// TwinCAT 3 PLC project RT1
// ProgramVersion: 3.1.4026.16
// libraries:
//   Tc2_ControllerToolbox, * (Beckhoff Automation GmbH)
//   Tc2_Standard, * (Beckhoff Automation GmbH)
//   Tc2_System, * (Beckhoff Automation GmbH)
//   Tc2_Utilities, * (Beckhoff Automation GmbH)
//   Tc3_Module, * (Beckhoff Automation GmbH)
//   VisuDialogs, * (System)
// project tree:
//   / GlobalTextList.TcGTLO, PlcTask.TcTTO, Visualization Manager.TcVMO (not stored)
//   POUs/AuxFuns/ FB_AutoResetBool.TcPOU, FB_Blink.TcPOU, FB_INC_DEC_Integer.TcPOU, FB_RangeMonitor.TcPOU, prgTestAuxsFuns.TcPOU
//   POUs/Conversion/ F_DtToSqlTime.TcPOU, F_DtToSqlTime2.TcPOU, F_DtToStr.TcPOU, F_LrealToExcel.TcPOU, F_MatIdtoStr.TcPOU, F_TimeStToFileStr.TcPOU
//   POUs/CO_Ntrollers/ FB_BasicHist.TcPOU, PIController.TcPOU
//   POUs/Filters/ FB_AvgFilter.TcPOU (not stored), FB_SignalGen.TcPOU, prgFilterTesting.TcPOU
//   POUs/ MAIN.TcPOU
//   POUs/Math/ betwenLimits.TcPOU, CharCurve.TcPOU, CheckDivZero.TcPOU, Derivative.TcPOU, DerivativeFiltered.TcPOU, DerivativeFiltered_2.TcPOU, FB_CalcKeyPoints.TcPOU, FB_CalcPeriod.TcPOU, FB_RampReal.TcPOU, FB_RMSCalc.TcPOU, FB_TimeBasedIntegrator.TcPOU, FB_TimeCounter.TcPOU, FirstDegResponse.TcPOU, F_AdjustDecimals.TcPOU, F_AdjustPrecision.TcPOU, F_SimpleDeadBand.TcPOU, GVL_Math.TcGVL, Integral.TcPOU, LinTrafoLimitLess.TcPOU, LinTrafo_1.TcPOU, prgMathTesting.TcPOU, SawTooth.TcPOU, TriangleWave.TcPOU
//   POUs/OrderAlgorithms/ F_SortBubble.TcPOU, F_SortInsertion.TcPOU
//   POUs/SignalCalc/ FB_RmsCalc2.TcPOU
//   POUs/SpecialTriggers/ FB_ChangeTrig.TcPOU, FB_Int_Trig.TcPOU, FB_Int_TrigFall.TcPOU, FB_Int_TrigRise.TcPOU, prgTrigTesting.TcPOU
//   POUs/Statistics/ FB_BasicStatsFuns.TcPOU, prgTestStatistics.TcPOU
//   VISUs/AuxScreens/ Footer.TcVIS
//   VISUs/ Math.TcVIS, Visualization.TcVIS
// real-time tasks:
//   TASK PlcTask: cycle T#10ms, priority 20, ADS port 350

CONFIGURATION RT1
    RESOURCE PLC ON TwinCAT3
        TASK PlcTask(INTERVAL := T#10ms, PRIORITY := 20);
        PROGRAM MAIN WITH PlcTask : MAIN;
    END_RESOURCE
END_CONFIGURATION

// ---- POUs/Math/GVL_Math.TcGVL
{attribute 'qualified_only'}
VAR_GLOBAL PERSISTENT
	rIntegratorResult:LREAL;
END_VAR

// ---- POUs/MAIN.TcPOU
PROGRAM MAIN
VAR

	sinGen:FB_CTRL_SIGNAL_GENERATOR;
	mode: Tc2_ControllerToolbox.E_CTRL_MODE := Tc2_ControllerToolbox.E_CTRL_MODE.eCTRL_MODE_ACTIVE;
	sine: LREAL;
	paramSin: Tc2_ControllerToolbox.ST_CTRL_SIGNAL_GENERATOR_PARAMS := (tCtrlCycleTime := TIME#10MS, tTaskCycleTime := TIME#10MS, eSignalType := E_CTRL_SIGNAL_TYPE.eCTRL_SINUS, tCylceDuration := TIME#500MS, fAmplitude := 2);
	rms1: FB_RMSCalc;
	rms2: FB_RmsCalc2;
	rmsOut1: LREAL;
	rmsOut2: LREAL;
	bResetRms: BOOL;
	rPeriod: LREAL := 1;
END_VAR

prgTrigTesting();
prgTestAuxsFuns();
prgTestStatistics();
prgFilterTesting();
prgMathTesting();


sinGen(
	fManValue:= , 
	eMode:=mode , 
	fOut=> sine, 
	eState=> , 
	eErrorId=> , 
	bError=> , 
	stParams:= paramSin);
	


rms1(
	rInput:= sine, 
	rPastTime:= 0.01, 
	bReset:= bResetRms, 
	rPeriod:=rPeriod , 
	rRmsValue=> rmsOut1);
	
rms2(in:= sine, timePerCycle:= 0.01, result=> rmsOut2);

END_PROGRAM

// ---- POUs/Math/FB_RMSCalc.TcPOU
FUNCTION_BLOCK FB_RMSCalc
VAR_INPUT
	rInput:LREAL;
	rPastTime:LREAL;
	bReset: BOOL;
	rPeriod: LREAL;
END_VAR
VAR_OUTPUT
	rRmsValue:LREAL;
END_VAR
VAR
	rmsIntegral:Integral;
END_VAR
(*Bloco funcional calcula o valor RMS de uma onda senoidal*)
(*Ha limitacoes quanto à frequencia utilizada (os testes foram feitos com frequencias de ate 12hz)*)
(*e quanto ao scan do plc (task de 2ms, mais baixas apresentam problemas)*)

IF bReset THEN
	rRmsValue:=SQRT(1/rPeriod *(rmsIntegral.rIntegral));
END_IF
rmsIntegral(rInput:=EXPT(rInput,2),rPastTime:=rPastTime , bReset:=bReset);

END_FUNCTION_BLOCK

// ---- POUs/Math/Integral.TcPOU
FUNCTION_BLOCK Integral
VAR_INPUT
	rInput:LREAL;		(*Valor de entrada*)
	rPastTime:LREAL;	(*tempo decorrido em Seg*)
	bReset: BOOL;	(*reinicia o bloco da integral*)
END_VAR
VAR_OUTPUT
	rIntegral:LREAL;	(*integral calculada*)
END_VAR
VAR
	rOldIntegral: LREAL;	(*Ultimo valor da integral*)
END_VAR
(*Este bloco funcional calcula a integral de uma funcao*)

IF bReset THEN
	rIntegral:=0;
	rOldIntegral:=0;
ELSE
	rIntegral:=rPastTime*rInput+rOldIntegral;
END_IF
rOldIntegral:=rIntegral;

END_FUNCTION_BLOCK

// ---- POUs/SignalCalc/FB_RmsCalc2.TcPOU
FUNCTION_BLOCK FB_RmsCalc2
VAR_INPUT
	in:LREAL;				//input sinal to calculate rms value
	timePerCycle:LREAL;		//time per cycle in seconds
END_VAR
VAR_OUTPUT
	result:LREAL;
END_VAR
VAR
	ar:ARRAY[1..100] OF LREAL;
	i: INT;
	sum,mean,t:LREAL;
END_VAR

FOR i:= 100 TO 2 BY -1 DO
	ar[i]:= ar[i-1];
END_FOR
ar[1]:=in;
sum:=0;

FOR i:= 1 TO 100 DO
	sum:=sum + EXPT(ar[i],2);
END_FOR
mean:= sum/100;
t:=100*timePerCycle;
result:= SQRT((1/t)*mean);

END_FUNCTION_BLOCK

// ---- POUs/SpecialTriggers/prgTrigTesting.TcPOU
PROGRAM prgTrigTesting
VAR
	changeTrig1:FB_ChangeTrig;
	udi:UDINT:=10;
	udiTrigCnt:UDINT;
	changeTrig2:FB_ChangeTrig;
	r1:REAL:=10;
	r1TrigCnt2:UDINT;
	changeTrigStr:FB_ChangeTrig;
	s1:STRING:='Boa tarde';
	sTringCnt:UDINT;
END_VAR

IF changeTrig1.M_ChngTrig(udi) THEN
	udiTrigCnt:=udiTrigCnt+1;
END_IF
IF changeTrig2.M_ChngTrig(in:= r1) THEN
	r1TrigCnt2:=r1TrigCnt2+1;
END_IF
IF changeTrigStr.M_ChngTrig(s1) THEN
	sTringcnt:=sTringcnt+1;
END_IF

END_PROGRAM

// ---- POUs/SpecialTriggers/FB_ChangeTrig.TcPOU
FUNCTION_BLOCK FB_ChangeTrig
VAR_INPUT
END_VAR
VAR_OUTPUT
END_VAR
VAR
	internalPointer:POINTER TO BYTE;
	aBytes:ARRAY[0..254] OF BYTE;
END_VAR

METHOD M_ChngTrig : BOOL
VAR_INPUT
	in:ANY;
END_VAR
IF THIS^.internalPointer <> 0 THEN
	M_ChngTrig:= memcmp(in.pValue,THIS^.internalPointer, in.diSize) <> 0;
	memcpy(THIS^.internalPointer,in.pValue,in.diSize);
ELSE
	THIS^.internalPointer:= ADR(THIS^.aBytes);
END_IF
END_METHOD

END_FUNCTION_BLOCK

// ---- POUs/AuxFuns/prgTestAuxsFuns.TcPOU
PROGRAM prgTestAuxsFuns
VAR
	blink:FB_Blink;
	rBlinkOn:LREAL:=0.5;
	rBlinkOff:LREAL:=0.3;
	bOutputBlink: BOOL;
END_VAR

blink(tON:= LREAL_TO_TIME(rBlinkOn*1000), tOff:=LREAL_TO_TIME(rBlinkOff*1000) , output=> bOutputBlink);

END_PROGRAM

// ---- POUs/AuxFuns/FB_Blink.TcPOU
FUNCTION_BLOCK FB_Blink
VAR_INPUT
	tON,tOff:TIME;
END_VAR
VAR_OUTPUT
	output:BOOL;
END_VAR
VAR
	timer:ton;
END_VAR

timer(IN:=NOT timer.Q);
IF timer.Q THEN
	IF output THEN
		timer.PT:=tOff;
	ELSE
		timer.PT:=tOn;
	END_IF
	output:= NOT output;
END_IF

END_FUNCTION_BLOCK

// ---- POUs/Statistics/prgTestStatistics.TcPOU
PROGRAM prgTestStatistics
VAR
	statistics:FB_BasicStatsFuns;
	aStats: ARRAY [1..7] OF LREAL := [15, 12, 11, 7, -5, 33, 45];
	avg: LREAL;
	maxi: LREAL;
	mini: LREAL;
	range: LREAL;
	variance: LREAL;
	std:LREAL;
END_VAR

avg:= statistics.M_Avg(aStats);

maxi:=statistics.M_Max(aStats);

mini:= statistics.M_Min(aStats);

range:= statistics.M_Range(aStats);

variance:=statistics.M_Variance(aStats);

std:= statistics.M_Std(aStats);

END_PROGRAM

// ---- POUs/Statistics/FB_BasicStatsFuns.TcPOU
FUNCTION_BLOCK FB_BasicStatsFuns
VAR_INPUT
END_VAR
VAR_OUTPUT
END_VAR
VAR
END_VAR

METHOD M_Avg : LREAL
VAR_IN_OUT
	a : ARRAY[*] OF LREAL;
END_VAR

VAR
	upper: DINT;
	lower: DINT;
	sum:LREAL;
	idx:DINT;
	qtt: LREAL;
	avg: LREAL;
END_VAR
upper:=UPPER_BOUND(a,1);
lower:=LOWER_BOUND(a,1);

qtt:= DINT_TO_LREAL(upper-lower+1);

sum:=0;
FOR idx:=lower TO upper DO
	sum:= sum + a[idx];
END_FOR
IF qtt <> 0 THEN
	avg:= sum/qtt;
END_IF
M_Avg:=avg;
END_METHOD

METHOD M_Max : LREAL
VAR_IN_OUT
	a:ARRAY[*] OF LREAL;
END_VAR
VAR
	maximum:LREAL;
	upper: DINT;
	lower: DINT;
	range: LREAL;
	idx: DINT;
END_VAR
upper:=UPPER_BOUND(a,1);
lower:=LOWER_BOUND(a,1);

range:= DINT_TO_LREAL(upper-lower+1);

maximum:= a[lower];

FOR idx:= lower TO upper DO
	maximum:= MAX(maximum, a[idx]);
END_FOR
M_Max:= maximum;
END_METHOD

METHOD M_Min : LREAL
VAR_IN_OUT
	a:ARRAY[*] OF LREAL;
END_VAR
VAR
	minimum:LREAL;
	upper: DINT;
	lower: DINT;
	range: LREAL;
	idx: DINT;	
END_VAR
upper:=UPPER_BOUND(a,1);
lower:=LOWER_BOUND(a,1);

range:= DINT_TO_LREAL(upper-lower+1);

minimum:= a[lower];

FOR idx:= lower TO upper DO
	minimum:= MIN(minimum, a[idx]);
END_FOR
M_Min:= minimum;
END_METHOD

METHOD M_Range : LREAL
VAR_IN_OUT
	a:ARRAY[*] OF LREAL;
END_VAR
VAR
	maximum, minimum, range:LREAL;
END_VAR
maximum:= M_Max(a);
minimum:= M_Min(a);

range:= maximum-minimum;
M_Range:= range;
END_METHOD

METHOD M_Std : LREAL
VAR_IN_OUT
	a : ARRAY[*] OF LREAL;
END_VAR
VAR
	variance:LREAL;
	std:LREAL;
END_VAR
variance:= M_Variance(a);
std:= SQRT(variance);
M_Std:=std;
END_METHOD

METHOD M_Variance : LREAL
VAR_IN_OUT
	a : ARRAY[*] OF LREAL;
END_VAR
VAR
	avg, qtt:lreal;
	upper: DINT;
	lower: DINT;
	idx: DINT;
	numerator:LREAL;
END_VAR
upper:=UPPER_BOUND(a,1);
lower:=LOWER_BOUND(a,1);

qtt:= DINT_TO_LREAL(upper-lower+1);

avg:=M_Avg(a);
numerator:=0;

FOR idx:= lower TO upper DO
	numerator:= numerator+ EXPT(a[idx]-avg,2);
END_FOR

IF qtt <> 0 THEN
	M_Variance:= numerator/qtt;
END_IF
END_METHOD

END_FUNCTION_BLOCK

// ---- POUs/Filters/prgFilterTesting.TcPOU
PROGRAM prgFilterTesting
VAR
	t:LREAL;
	squareSignal:LREAL;
	valueAdd:LREAL:=0.01;
END_VAR

t:= t+valueAdd;

squareSignal:= SIN(t) + SIN(3*t)/3+ SIN(5*t)/5 + SIN(7*t)/7 + SIN(9*t)/9;

END_PROGRAM

// ---- POUs/Math/prgMathTesting.TcPOU
PROGRAM prgMathTesting
VAR
	noise:FB_CTRL_NOISE_GENERATOR;
	mode: E_CTRL_MODE := E_CTRL_MODE.eCTRL_MODE_ACTIVE;
	paramNoise: ST_CTRL_NOISE_GENERATOR_PARAMS := (tCtrlCycleTime := TIME#10MS, tTaskCycleTime := TIME#10MS, fAmplitude := 5);
	integrator:FB_TimeBasedIntegrator;
	addNegative: BOOL;
END_VAR

noise(
	fManSyncValue:= , 
	eMode:= mode, 
	fOut=> , 
	eState=> , 
	eErrorId=> , 
	bError=> , 
	stParams:= paramNoise);

integrator(
	tBaseTime:= T#1S, 
	rIn:= noise.fOut, 
	addNegativeValues:= addNegative, 
	bErr=> , 
	rAccumulator:= GVL_math.rIntegratorResult);

END_PROGRAM

// ---- POUs/Math/FB_TimeBasedIntegrator.TcPOU
FUNCTION_BLOCK FB_TimeBasedIntegrator
VAR_INPUT
	tBaseTime:TIME:=T#1S;
	rIn:LREAL;
	addNegativeValues:BOOL;
	reset:BOOL;
END_VAR
VAR_OUTPUT
	bErr: BOOL;
END_VAR
VAR
	t1:TON;
END_VAR
VAR_IN_OUT
	rAccumulator:LREAL;
END_VAR

IF tBaseTime = T#0S THEN
	RETURN;
END_IF

t1(IN:= NOT t1.Q, PT:= tBaseTime);

IF t1.Q AND addNegativeValues THEN
	rAccumulator:=rAccumulator+rIn;
ELSIF t1.Q AND NOT addNegativeValues THEN
	rAccumulator := SEL(rIn >0, rAccumulator, rAccumulator+rIn);
END_IF

IF reset THEN
	rAccumulator:=0;
END_IF

END_FUNCTION_BLOCK

// ---- POUs/AuxFuns/FB_AutoResetBool.TcPOU
FUNCTION_BLOCK FB_AutoResetBool
VAR_INPUT
	tResetTime:TIME:=T#100MS;
END_VAR
VAR_OUTPUT
END_VAR
VAR
	t1:TON;
END_VAR
VAR_IN_OUT
	bReset: BOOL;
END_VAR

t1(IN:=bReset , PT:= tResetTime);
IF t1.Q THEN
	bReset:=FALSE;
END_IF

END_FUNCTION_BLOCK

// ---- POUs/AuxFuns/FB_INC_DEC_Integer.TcPOU
FUNCTION_BLOCK FB_INC_DEC_Integer
VAR_INPUT
	bIncrease: BOOL;
	bDecrease: BOOL;
	iMaxValue:INT;
	iMinValue:INT;
END_VAR
VAR_OUTPUT
END_VAR
VAR
	IncreaseR_TRIG:R_TRIG;
	DecreaseR_TRIG:R_TRIG;
END_VAR
VAR_IN_OUT
	iVariable:INT;
END_VAR

IncreaseR_TRIG(CLK:= bIncrease);
DecreaseR_TRIG(CLK:=bDecrease );

IF IncreaseR_TRIG.Q AND iVariable<iMaxValue THEN
	iVariable:=iVariable+1;
END_IF
IF DecreaseR_TRIG.Q  AND iVariable>iMinValue THEN
	iVariable:=iVariable-1;
END_IF

END_FUNCTION_BLOCK

// ---- POUs/AuxFuns/FB_RangeMonitor.TcPOU
FUNCTION_BLOCK FB_RangeMonitor
VAR_INPUT
	rIn,rMax,rMin:LREAL;
	tTimeFilter:TIME;
	bReset: BOOL;

END_VAR
VAR_OUTPUT
	bOut:BOOL;
END_VAR
VAR
	t1:TON;
END_VAR


t1(IN:=rIn>rMax OR rIn<rMin , PT:= tTimeFilter);

IF t1.Q AND NOT bReset THEN
	bOut:=TRUE;
ELSIF bReset THEN
	bOut:=FALSE;	
END_IF

END_FUNCTION_BLOCK

// ---- POUs/Conversion/F_DtToSqlTime.TcPOU
FUNCTION F_DtToSqlTime : STRING
VAR_INPUT
	dtIn:TIMESTRUCT;
END_VAR
VAR
	s1:STRING;
END_VAR

s1:= WORD_TO_STRING(dtIn.wYear);
s1:=CONCAT(S1,'-');
S1:=CONCAT(S1,WORD_TO_STRING(dtIn.wMonth));
s1:=CONCAT(s1,'-');
s1:=CONCAT(S1,WORD_TO_STRING(dtIn.wDay));
s1:=CONCAT(s1,' ');
s1:=CONCAT(s1,WORD_TO_STRING(dtIN.wHour));
s1:=CONCAT(S1,':');
S1:=CONCAT(s1,WORD_TO_STRING(dtIN.wMinute));
s1:=CONCAT(s1,':');
s1:=CONCAT(s1,WORD_TO_STRING(dtIN.wSecond));

F_DtToSqlTime:=S1;

END_FUNCTION

// ---- POUs/Conversion/F_DtToSqlTime2.TcPOU
FUNCTION F_DtToSqlTime2 : STRING
VAR_INPUT
	dtIn:TIMESTRUCT;
END_VAR
VAR
	s1:STRING;
END_VAR

s1:= WORD_TO_STRING(dtIn.wYear);
//s1:=CONCAT(S1,'-');
IF dtIn.wMonth<10 THEN
	S1:=CONCAT(S1,'0');
	S1:=CONCAT(S1,WORD_TO_STRING(dtIn.wMonth));
ELSE
	S1:=CONCAT(S1,WORD_TO_STRING(dtIn.wMonth));
END_IF
//s1:=CONCAT(s1,'-');
IF dtIn.wDay<10 THEN
	S1:=CONCAT(S1,'0');
	s1:=CONCAT(S1,WORD_TO_STRING(dtIn.wDay));
ELSE
	s1:=CONCAT(S1,WORD_TO_STRING(dtIn.wDay));
END_IF
s1:=CONCAT(s1,' ');
s1:=CONCAT(s1,WORD_TO_STRING(dtIN.wHour));
s1:=CONCAT(S1,':');
S1:=CONCAT(s1,WORD_TO_STRING(dtIN.wMinute));
s1:=CONCAT(s1,':');
s1:=CONCAT(s1,WORD_TO_STRING(dtIN.wSecond));

F_DtToSqlTime2:=S1;

END_FUNCTION

// ---- POUs/Conversion/F_DtToStr.TcPOU
FUNCTION F_DtToStr : STRING
VAR_INPUT
	dt1:DT;
END_VAR
VAR
	s1:STRING;
	t1:TIMESTRUCT;
END_VAR

t1:=DT_TO_SYSTEMTIME(dt1);
s1:=WORD_TO_STRING(t1.wDay);
s1:= CONCAT(S1,'/');
S1:=CONCAT(s1,WORD_TO_STRING(t1.wMonth));
s1:=CONCAT(s1,'/');
s1:=CONCAT(s1,WORD_TO_STRING(t1.wYear));
s1:=CONCAT(s1,' ');
s1:=CONCAT(s1,WORD_TO_STRING(t1.wHour));
s1:=CONCAT(s1,':');
s1:=CONCAT(s1,WORD_TO_STRING(t1.wMinute));
s1:=CONCAT(s1,':');
s1:=CONCAT(s1, WORD_TO_STRING(t1.wSecond));
F_DtToStr:=s1;

END_FUNCTION

// ---- POUs/Conversion/F_LrealToExcel.TcPOU
FUNCTION F_LrealToExcel : STRING
VAR_INPUT
	bUseComma: BOOL;
	r1:LREAL;
END_VAR
VAR
	s1:STRING;
	pos: INT;
END_VAR

//in portuguese Excel should have a comma instead of a dot
s1:=LREAL_TO_STRING(r1);
IF bUseComma THEN
	pos:= find(s1,'.');
	IF pos <> 0 THEN
		s1:=replace(s1,',',1,pos);
	END_IF	
END_IF

F_LrealToExcel:=s1;

END_FUNCTION

// ---- POUs/Conversion/F_MatIdtoStr.TcPOU
FUNCTION F_MatIdtoStr : STRING(20)
VAR_INPUT
	materialId:DINT;
END_VAR
VAR
	i:UINT;
	s1: STRING;
END_VAR

FOR i :=1 TO GVLConst.uiLastMaterialPossible DO
	IF G_DBConn.aMaterialAvailable[i].ID = materialId AND materialId <> 0 THEN
		s1:=G_Dbconn.aMaterialAvailable[i].matId;
		EXIT;
	ELSIF materialId =  0 THEN
		s1:='';
		EXIT;
	END_IF
END_FOR
F_MatIdtoStr:=s1;

END_FUNCTION

// ---- POUs/Conversion/F_TimeStToFileStr.TcPOU
FUNCTION F_TimeStToFileStr : STRING
VAR_INPUT
	timeToConvert:TIMESTRUCT;
END_VAR
VAR
	s1:STRING;
END_VAR
//Converts a timestruct variable to a string that can be used as file name

s1:=WORD_TO_STRING(timeToConvert.wYear);
s1:=CONCAT(s1,WORD_TO_STRING(timeToConvert.wMonth));
s1:=CONCAT(s1,WORD_TO_STRING(timeToConvert.wDay));
s1:=CONCAT(s1,'_');
s1:=CONCAT(s1,WORD_TO_STRING(timeToConvert.wHour));
s1:=CONCAT(s1,'_');
s1:=CONCAT(s1,WORD_TO_STRING(timeToConvert.wMinute));
s1:=CONCAT(s1,'_');
s1:=CONCAT(s1,WORD_TO_STRING(timeToConvert.wSecond));

F_TimeStToFileStr:=s1;

END_FUNCTION

// ---- POUs/CO_Ntrollers/FB_BasicHist.TcPOU
FUNCTION_BLOCK FB_BasicHist
VAR_INPUT
	fHisteresis,fDesiredValue,fActualValue:LREAL;
END_VAR
VAR_OUTPUT
	output,error:BOOL;
END_VAR
VAR
	maximum: LREAL;
	minimum: LREAL;
	trigMaxReached, trigMinReached:R_TRIG;
END_VAR

IF fHisteresis>0 THEN
	error:=FALSE;
	//
	maximum:=fDesiredValue + fHisteresis/2;
	minimum:= fDesiredValue-fHisteresis/2;
	trigMaxReached(CLK:=fActualValue>maximum);
	trigMinReached(CLK:= fActualValue<minimum);
	IF trigMaxReached.Q THEN
		output:=TRUE;
	END_IF
	IF trigMinReached.Q THEN
		output:=FALSE;
	END_IF
ELSE
	output:=FALSE;
	error:=TRUE;	
END_IF

END_FUNCTION_BLOCK

// ---- POUs/CO_Ntrollers/PIController.TcPOU
FUNCTION_BLOCK PIController
VAR_INPUT
	Kp:LREAL;				(*Ganho proporcional*)
	Ki:LREAL;				(*Ganho integral*)
	rSp:LREAL;				(*Set point*)
	rPv:LREAL;				(*Process Value*)
	rPastTime:LREAL;			(*tempo decorrido em segundos*)
	rLowerSaturation:LREAL;	(*Valor minimo que e sai do controlador*)
	rUpperSaturation:LREAL;	(*Valor maximo que sai do controlador*)
	bReset:BOOL;			(*Reset do controlador*)
END_VAR
VAR_OUTPUT
	rOutput:LREAL;			(*saida do controlador*)
END_VAR
VAR
	Integrator:Integral;			(*bloco calcula o sinla integral*)
	rError: LREAL;			(*sinal de erro*)
END_VAR

(*Calcula o sinal de erro*)
rError:=rSp -rPv;
(*Calcula a parte integral*)
Integrator(rInput:=rError , rPastTime:= rPastTime, bReset:=bReset );

rOutput:= LIMIT(rLowerSaturation,Kp*rError+Ki*Integrator.rIntegral,rUpperSaturation);

END_FUNCTION_BLOCK

// ---- POUs/Filters/FB_SignalGen.TcPOU
FUNCTION_BLOCK FB_SignalGen
VAR_INPUT
END_VAR
VAR_OUTPUT
END_VAR
VAR
END_VAR

END_FUNCTION_BLOCK

// ---- POUs/Math/betwenLimits.TcPOU
FUNCTION betwenLimits : BOOL
VAR_INPUT
	rLower:REAL;			(*limite inferior*)
	rInput:REAL;			(*entrada*)
	rUpper:REAL;			(*Limite superior*)
END_VAR
VAR
END_VAR
(*Esta funcao retorna true caso a entrada esteja entre os limites rLower e rUpper*)
(*Nao importando se o Lower e maior ou menor que o upper*)

betwenLimits:=(rInput>=rLower) AND (rInput<=rUpper) OR  (rInput<=rLower) AND (rInput>=rUpper);

END_FUNCTION

// ---- POUs/Math/CharCurve.TcPOU
FUNCTION_BLOCK CharCurve
VAR_INPUT
	rInput:REAL;		(*entrada a ser linearizada*)
	Lintab:tsLintab;	(*tabela de linearizacao*)
END_VAR
VAR_OUTPUT
	rOutPut:REAL;	(*saida linearizada*)
END_VAR
VAR
	i: INT;			(*auxiliar de contagem*)
END_VAR
(*Gera linearizacao da entrada atraves da tabela de Lintab*)
(*aplicam-se valores positivos*)

FOR i:= 1 TO Lintab.iNumOfPoints DO
	IF rInput>Lintab.Point[i-1].rX AND rInput<=Lintab.Point[i].rX THEN
		EXIT;
	END_IF
END_FOR
IF i<=Lintab.iNumOfPoints THEN
	rOutPut:=Lintab.Point[i-1].rY+ LinTrafoLimitLess(rInput-Lintab.Point[i-1].rX,Lintab.Point[i-1].rX,Lintab.Point[i].rX,0,Lintab.Point[i].rY-Lintab.Point[i-1].rY);
ELSE
	rOutPut:=0;
END_IF

END_FUNCTION_BLOCK

// ---- POUs/Math/LinTrafoLimitLess.TcPOU
FUNCTION LinTrafoLimitLess : REAL
VAR_INPUT
	rValue:REAL;			(*Valor a sofrer escala*)
	rInMin:REAL;			(*Valor minimo de entrada*)
	rInMax:REAL;			(*valor Maximo de entrada*)
	rOutMin:REAL;		(*Valor minimo da saida*)
	rOutMax:REAL;		(*Valor maximo de saida*)
END_VAR
VAR
END_VAR
(*Esta funcao admite tanto valores negativos quanto positivos (porem a saida so sera negativa se o valor de entrada for negativo)*)

(*Realiza uma simples escala*)
LinTrafoLimitLess:=rValue*(rOutMax-rOutMin)/CheckDivZero(rInMax-rInMin);

END_FUNCTION

// ---- POUs/Math/CheckDivZero.TcPOU
FUNCTION CheckDivZero : REAL
VAR_INPUT
	rInput:REAL;	(*Entrada a ser comparada*)
END_VAR
VAR
END_VAR
(*Apenas verifica se a entrada e igual a zero para poder realizar um divisao*)
(*just check if the input is zero to make a division operation*)

(*Apenas verifica se a entrada dessa funcao é igual a zero*)
IF rInput <> 0 THEN
	CheckDivZero := rInput;
ELSE
	CheckDivZero:=1;
END_IF

END_FUNCTION

// ---- POUs/Math/Derivative.TcPOU
FUNCTION_BLOCK Derivative
VAR_INPUT
	rValue:LREAL;			(*Valor a ser derivado*)
	rPastTime:LREAL;		(*tempo decorrido em ms*)
END_VAR
VAR_OUTPUT
	rDerivative:LREAL;		(*valor derivado*)
END_VAR
VAR
	rOldValue: LREAL;
END_VAR

IF rPastTime>0 THEN
	rDerivative:=(rValue-rOldValue)/rPastTime;
ELSE
	rDerivative:=0;
END_IF
rOldValue:=rValue;

END_FUNCTION_BLOCK

// ---- POUs/Math/DerivativeFiltered.TcPOU
FUNCTION_BLOCK DerivativeFiltered
VAR_INPUT
	rValue:LREAL;					(*Valor a ser derivado*)
	tFilterTime:TIME;				(*Tempo a considerar no filtro derivativo*)
END_VAR
VAR_OUTPUT
	rDerivative:LREAL;				(*valor derivado*)
END_VAR
VAR
	rOldValue: LREAL;
	TimeCounter: FB_TimeCounter;	(*Conta o tempo para o filtro da derivada*)
END_VAR
(*Calcula a derivada baseado num tempo estabelecido na variavel *)

TimeCounter(tIn:=tFilterTime);
(*rPastTime:=;*)
IF tFilterTime>t#0ms AND TimeCounter.bOutPulse THEN
	rDerivative:=(rValue-rOldValue)/(TIME_TO_LREAL(tFilterTime)/1000);
	rOldValue:=rValue;
ELSIF tFilterTime=t#0ms THEN
	rDerivative:=0;
END_IF

END_FUNCTION_BLOCK

// ---- POUs/Math/FB_TimeCounter.TcPOU
FUNCTION_BLOCK FB_TimeCounter
VAR_INPUT
	tIn: TIME;
END_VAR
VAR_OUTPUT
	bOutPulse: BOOL;
END_VAR
VAR
	timer_01: TON;
END_VAR

(*Este bloco funcional fornece um pulso na saida a cada período de tempo pre determinado*)
timer_01(IN:= NOT timer_01.Q , PT:= tIn , Q=>bOutPulse , ET=> );

END_FUNCTION_BLOCK

// ---- POUs/Math/DerivativeFiltered_2.TcPOU
FUNCTION_BLOCK DerivativeFiltered_2
VAR_INPUT
	rValue:LREAL;			(*Valor a ser derivado*)
	rPastTime:LREAL;		(*tempo decorrido em ms*)
	iNumOfCycles:INT:=4;
END_VAR
VAR_OUTPUT
	rDerivative:LREAL;		(*valor derivado*)
END_VAR
VAR
	rOldValue: LREAL;
	rTimeToCalc:LREAL;
	iPastCycles:INT;
END_VAR

iPastCycles:=iPastCycles+1;
IF iPastCycles<iNumOfCycles OR (iNumOfCycles<=0) THEN
	RETURN;
ELSE
	iPastCycles:=0;
END_IF
IF rPastTime>0 THEN
	rDerivative:=(rValue-rOldValue)/(rPastTime*INT_TO_LREAL(iNumOfCycles));
ELSE
	rDerivative:=0;
END_IF
rOldValue:=rValue;

END_FUNCTION_BLOCK

// ---- POUs/Math/FB_CalcKeyPoints.TcPOU
FUNCTION_BLOCK FB_CalcKeyPoints
VAR_INPUT
	bStartNow:BOOL;
	rInY,rInX:LREAL;
	rPointGiven:LREAL;
	rToleranceGiven:LREAL:=0.1;
END_VAR
VAR_OUTPUT
	rMin:LREAL;
	rMax:LREAL;
	rGivenPointY:LREAL;
END_VAR
VAR
	startNowR_TRIG:R_TRIG;
	givenPointR_TRIG:R_TRIG;
	rInternalMin:LREAL;
END_VAR

startNowR_TRIG(CLK:=bStartNow);
IF startNowR_TRIG.Q THEN
	rMax:=0;
	rMin:=0;
	rGivenPointY:=0;
	rInternalMin:=0;
END_IF
IF bStartNow THEN
	rMax:=MAX(rMax,rInY);
	rInternalMin:=MIN(rInternalMin,rInY);	
END_IF

givenPointR_TRIG(CLK:=betwenLimits(rPointGiven-rToleranceGiven,rInX,rPointGiven+rToleranceGiven));
IF givenPointR_TRIG.Q THEN
	rMin:=rInternalMin;
	rGivenPointY:=rInY;
END_IF

END_FUNCTION_BLOCK

// ---- POUs/Math/FB_CalcPeriod.TcPOU
FUNCTION_BLOCK FB_CalcPeriod
VAR_INPUT
	rWave:LREAL;
	rDCValue:LREAL;	(*distancia entre 0 e o valor medio da onda (Valor DC)*)
END_VAR
VAR_OUTPUT
	rPeriod: LREAL;
	bNewStarted:BOOL;
END_VAR
VAR
	newWaveStartedR_TRIG:R_TRIG;
	rRelativeInput: LREAL;
	rOldRelativeInput: LREAL;
	periodTON:TON;
END_VAR
(*Este bloco funcional tem por objetivo calcular o periodo de uma onda senoidal*)
(*Dada a entrada o mesmo fornece: o periodo(rPeriod) e um borda de subida na variavel (bNewPeriodStarted)*)
(*Toda vez que um novo periodo é iniciado*)

rRelativeInput:=rWave-rDCValue;
newWaveStartedR_TRIG(CLK:=(rRelativeInput>0) AND (rOldRelativeInput <0));
rOldRelativeInput:=rRelativeInput;
IF newWaveStartedR_TRIG.Q THEN
	rPeriod:=TIME_TO_LREAL(periodTON.ET)/1000;
END_IF
periodTON(IN:=NOT newWaveStartedR_TRIG.Q , PT:=t#1d);
bNewStarted:=newWaveStartedR_TRIG.Q;

END_FUNCTION_BLOCK

// ---- POUs/Math/FB_RampReal.TcPOU
FUNCTION_BLOCK FB_RampReal
VAR_INPUT
	rValue,rRamp:LREAL;	(*Valor para rampear*)
	bEnable: BOOL;		(*habilita o funcionamento da rampa*)
	rTolerance: LREAL;	(*Tolerancia para considerar que a saida esta igual ao valor setado*)
END_VAR
VAR_OUTPUT
	rOutPut:LREAL;		(*valor calculado*)
	bInvalidValue: BOOL;	(*caso algum valor negativo seja inserido*)
END_VAR
VAR
	rampTON:TON;		(*Temporizador do gerador de rampas*)
	rOldValue: LREAL;		(*ultimo valor colocado na saida*)
END_VAR
(*Bloco gera saida rampeada de acordo com os valores fornecidos em rValue,rRamp e bEnable*)
(*So admite valores positivos, tanto para valores quanto para rampas, caso contrario gera um sinal de erro*)

IF rValue>=0 AND rRamp>=0 THEN
(*define o valor de tempo a ser utilizado na rampa*)
	IF rValue <> rOutPut AND bEnable THEN
		IF rValue > rOldValue THEN
			rampTON.PT:=LREAL_TO_TIME((rValue-rOldValue)*1000/CheckDivZero(rRamp));
		ELSIF rValue < rOldValue THEN
			rampTON.PT:=LREAL_TO_TIME((rOldValue-rValue)*1000/CheckDivZero(rRamp));
		ELSE
			rampTON.PT:=t#0s;
		END_IF
	ELSIF NOT bEnable THEN
		rOldValue:=0;
		rOutPut:=0;
	END_IF
	(*calcula o valor a ser somado/subtraido da rampa*)
	IF betwenLimits(rValue-rTolerance,rOutPut,rValue+rTolerance) THEN
		rOldValue:=rOutPut;
	END_IF
	(*temporizador utilizado para gerar as rampas*)
	rampTON(IN:= bEnable AND  rValue <> rOutPut );
	(*Calcula o valor de saida de acordo com os criterios pertinentes*)
	IF rValue > rOldValue THEN
		rOutPut:=LIMIT(0,(TIME_TO_LREAL(rampTON.ET)/1000)*rRamp+rOldValue,rValue);
	ELSIF rValue < rOldValue THEN
		rOutPut:=LIMIT(rValue,rOldValue-(TIME_TO_LREAL(rampTON.ET)/1000)*rRamp,rOldValue);
	ELSE
		rOutPut:=rValue;
	END_IF
	bInvalidValue:=FALSE;
ELSE
	rOutPut:=0;
	bInvalidValue:=TRUE;
END_IF

END_FUNCTION_BLOCK

// ---- POUs/Math/FirstDegResponse.TcPOU
FUNCTION_BLOCK FirstDegResponse
VAR_INPUT
	rTime:REAL;			(*Time current*)
	rDec:REAL;			(*Coeficient*)
	rInput:REAL;		(*Degree input*)
END_VAR
VAR_OUTPUT
	rOutput:REAL;
END_VAR
VAR
END_VAR

rOutput:= rInput*(1-EXPT(2.71,-rTime*rDec));

END_FUNCTION_BLOCK

// ---- POUs/Math/F_AdjustDecimals.TcPOU
FUNCTION F_AdjustDecimals : LREAL
VAR_INPUT
	rIn:LREAL;
	iPrecision:UINT:=2;
END_VAR
VAR
	rInternal: LREAL;
END_VAR


IF rIn <> 0 AND iPrecision<>0 THEN
	rInternal:=rIn*EXPT(10,iPrecision);
	rInternal:=FLOOR(rInternal);
	F_AdjustDecimals:=rInternal/EXPT(10,iPrecision);
ELSE 
	F_AdjustDecimals:=0;	
END_IF

END_FUNCTION

// ---- POUs/Math/F_AdjustPrecision.TcPOU
FUNCTION F_AdjustPrecision : LREAL (*Ajusta a precisao dos numeros em ponto flutuante*)
VAR_INPUT
	in:LREAL;
	iPrecision:INT;
END_VAR
VAR
END_VAR

F_AdjustPrecision:= SEL(in<0,FLOOR(in*EXPT(10,iPrecision))/EXPT(10,iPrecision),-FLOOR(ABS(in)*EXPT(10,iPrecision))/EXPT(10,iPrecision));

END_FUNCTION

// ---- POUs/Math/F_SimpleDeadBand.TcPOU
FUNCTION F_SimpleDeadBand : BOOL
VAR_INPUT
	rActualValue:REAL;		(*Actual Value measured*)
	rTolerance:REAL;			(*measurement Tolerance*)
	rReferenceValue:REAL;	(*Reference value*)
END_VAR
VAR
END_VAR

(*Dead Band calculation according to the given parameters*)
F_SimpleDeadBand:= betwenLimits(rReferenceValue-rTolerance, rActualValue, rReferenceValue+rTolerance);

END_FUNCTION

// ---- POUs/Math/LinTrafo_1.TcPOU
FUNCTION LinTrafo_1 : REAL
VAR_INPUT
	rValue:REAL;			(*Valor a sofrer escala*)
	rInMin:REAL;			(*Valor minimo de entrada*)
	rInMax:REAL;			(*valor Maximo de entrada*)
	rOutMin:REAL;		(*Valor minimo da saida*)
	rOutMax:REAL;		(*Valor maximo de saida*)
END_VAR
VAR
END_VAR
(*Esta funcao admite tanto valores negativos quanto positivos (porem a saida so sera negativa se o valor de entrada for negativo)*)

IF (rInMax-rInMin) <> 0 THEN
	LinTrafo_1:=rValue * (rOutMax-rOutMin)/ (rInMax-rInMin)+rOutMin;
END_IF

END_FUNCTION

// ---- POUs/Math/SawTooth.TcPOU
FUNCTION_BLOCK SawTooth
VAR_INPUT
	rPeriod:LREAL;		(*Periodo da onda dente de serra em segundos (so sao permitidos valores positivos)*)
	rAmplitude:LREAL;		(*Amplitude maxima da onda dente de serra (so sao permitidos valores positivos)*)
	bStart: BOOL;			(*inicia a geracao da onda*)
END_VAR
VAR_OUTPUT
	rOutPut: LREAL;		(*Sinal de saida*)
END_VAR
VAR
	sawToothTON: TON;		(*Conta o tempo de subida da onda dente de serra*)
END_VAR
(*Este bloco funcional gera uma onda dente de serra, na qual e possivel determinar o periodo e a maxima amplitude do sinal*)

IF (rPeriod>0) AND rAmplitude>0 THEN
	sawToothTON(IN:=bStart AND NOT sawToothTON.Q,PT:=REAL_TO_TIME(rPeriod*1000));
	rOutPut:=( TIME_TO_REAL(sawToothTON.ET)/1000)*rAmplitude/CheckDivZero(rPeriod);
ELSE
	rOutPut:=0;
END_IF

END_FUNCTION_BLOCK

// ---- POUs/Math/TriangleWave.TcPOU
FUNCTION_BLOCK TriangleWave
VAR_INPUT
	rAmplitude:REAL;		(*Amplitude da onda triangular (valor deve ser maior que zero)*)
	rRisingtime:REAL;		(*Tempo de subida da onda triangular em segundos*)
	rFallingTime:REAL;	(*Tempo de descida da onda triangular em segundos*)
	bStart:BOOL;			(*inicia geracao da onda*)
END_VAR
VAR_OUTPUT
	rOutput:REAL;			(*Saida da onda triangular*)
END_VAR
VAR
	rising: SawTooth;
	falling: SawTooth;
	i: INT := 1;
END_VAR

IF rAmplitude>0 THEN
	CASE i OF
	1:
		rising(rPeriod:= rRisingtime, rAmplitude:= rAmplitude, bStart:=bStart , rOutPut=>rOutput );
		IF rising.rOutPut = rAmplitude THEN
			i:=2;
		END_IF
	2:
		falling(rPeriod:= rFallingTime, rAmplitude:=rAmplitude , bStart:= bStart, rOutPut=> );
		rOutput:=rAmplitude- falling.rOutPut;
		IF falling.rOutPut = rAmplitude THEN
			rOutput:=0;
			i:=1;
		END_IF
	END_CASE
ELSE
	rOutput:=0;
END_IF

END_FUNCTION_BLOCK

// ---- POUs/OrderAlgorithms/F_SortBubble.TcPOU
FUNCTION F_SortBubble : BOOL
VAR_INPUT
	pArToSort: POINTER TO ARRAY[cFirstSortingElement..cLastSortingElement] OF LREAL;
	bSortUpDown: BOOL;		(*Classifica de maneira decrescente*)
END_VAR
VAR
	i: UINT;
	j: UINT;
	aux: LREAL;
END_VAR

IF bSortUpDown THEN
	FOR i:= cFirstSortingElement TO cLastSortingElement DO
		FOR j:=cFirstSortingElement TO (cLastSortingElement-1) DO
			IF pArToSort^[j] < pArToSort^[j+1] THEN
				aux := pArToSort^[j];
				pArToSort^[j] := pArToSort^[j+1];
				pArToSort^[j+1] := aux;
			END_IF
		END_FOR
	END_FOR
ELSE
	FOR i:= cFirstSortingElement TO cLastSortingElement DO
		FOR j:=cFirstSortingElement TO (cLastSortingElement-1) DO
			IF pArToSort^[j] > pArToSort^[j+1] THEN
				aux := pArToSort^[j];
				pArToSort^[j] := pArToSort^[j+1];
				pArToSort^[j+1] := aux;
			END_IF
		END_FOR
	END_FOR
END_IF

END_FUNCTION

// ---- POUs/OrderAlgorithms/F_SortInsertion.TcPOU
FUNCTION F_SortInsertion : BOOL
VAR_INPUT
	pArToSort: POINTER TO ARRAY[cFirstSortingElement..cLastSortingElement] OF LREAL;
	bSortUpDown: BOOL;		(*Classifica de maneira decrescente*)
END_VAR
VAR
	i,j:INT;
	eleito:LREAL;
END_VAR

IF NOT bSortUpDown THEN			(*inicia uma classificacao crescente*)
	FOR i:= cFirstSortingElement TO cLastSortingElement DO
		eleito:= pArToSort^[i];
		j:=i-1;
		WHILE ((j>0) AND (eleito < pArToSort^[j])) DO
			pArToSort^[j+1] :=pArToSort^[j];
			j:=j-1;
		END_WHILE
		pArToSort^[j+1]:=eleito;
	END_FOR
ELSE								(*Caso classificacao decrescente*)
	FOR i:= cFirstSortingElement TO cLastSortingElement DO
		eleito:= pArToSort^[i];
		j:=i-1;
		WHILE ((j>0) AND (eleito > pArToSort^[j])) DO
			pArToSort^[j+1] :=pArToSort^[j];
			j:=j-1;
		END_WHILE
		pArToSort^[j+1]:=eleito;
	END_FOR
END_IF

END_FUNCTION

// ---- POUs/SpecialTriggers/FB_Int_Trig.TcPOU
FUNCTION_BLOCK FB_Int_Trig
VAR_INPUT
	IN:INT;
END_VAR
VAR_OUTPUT
	Q:BOOL;
END_VAR
VAR
	M:INT;
END_VAR
(*neste bloco funcional a saida Q e ativa durante um ciclo toda vez que ocorre uma mudanca na variavel IN*)

Q:=IN<>M;
M:=IN;

END_FUNCTION_BLOCK

// ---- POUs/SpecialTriggers/FB_Int_TrigFall.TcPOU
FUNCTION_BLOCK FB_Int_TrigFall
VAR_INPUT
	IN:INT;
	inRequired:INT;
END_VAR
VAR_OUTPUT
	Q:BOOL;
END_VAR
VAR
	M:INT;
END_VAR
(*neste bloco funcional a saida Q e ativa durante um ciclo toda vez que IN se torna diferente a inRequired*)

Q:=(IN <> inRequired) AND (inRequired = M);
M:=IN;

END_FUNCTION_BLOCK

// ---- POUs/SpecialTriggers/FB_Int_TrigRise.TcPOU
FUNCTION_BLOCK FB_Int_TrigRise
VAR_INPUT
	IN:INT;
	inRequired:INT;
END_VAR
VAR_OUTPUT
	Q:BOOL;
END_VAR
VAR
	M:INT;
END_VAR
(*neste bloco funcional a saida Q e ativa durante um ciclo toda vez que IN se torna igual a inRequired*)

Q:=(IN=inRequired) AND (IN <> M);
M:=IN;

END_FUNCTION_BLOCK

// ---- GlobalTextList.TcGTLO
TEXTLIST GlobalTextList
  21 = '%.1f'
  493 = 'Blink'
  145 = 'MAIN'
  460 = 'MATH'
  96 = 'Off'
  963 = 'On'
END_TEXTLIST

// ---- VISUs/AuxScreens/Footer.TcVIS
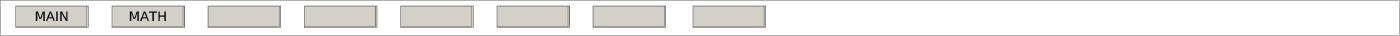
VISUALIZATION Footer  // 1920x50
    Button (21,8 100x30), "MAIN"
        OnMouseClick: change screen: Visualization
    Button (153,8 100x30), "MATH"
    Button (285,8 100x30)
    Button (417,8 100x30)
    Button (549,8 100x30)
    Button (681,8 100x30)
    Button (813,8 100x30)
    Button (950,8 100x30)
END_VISUALIZATION

// ---- VISUs/Math.TcVIS
VISUALIZATION Math  // 1920x1080
END_VISUALIZATION

// ---- VISUs/Visualization.TcVIS
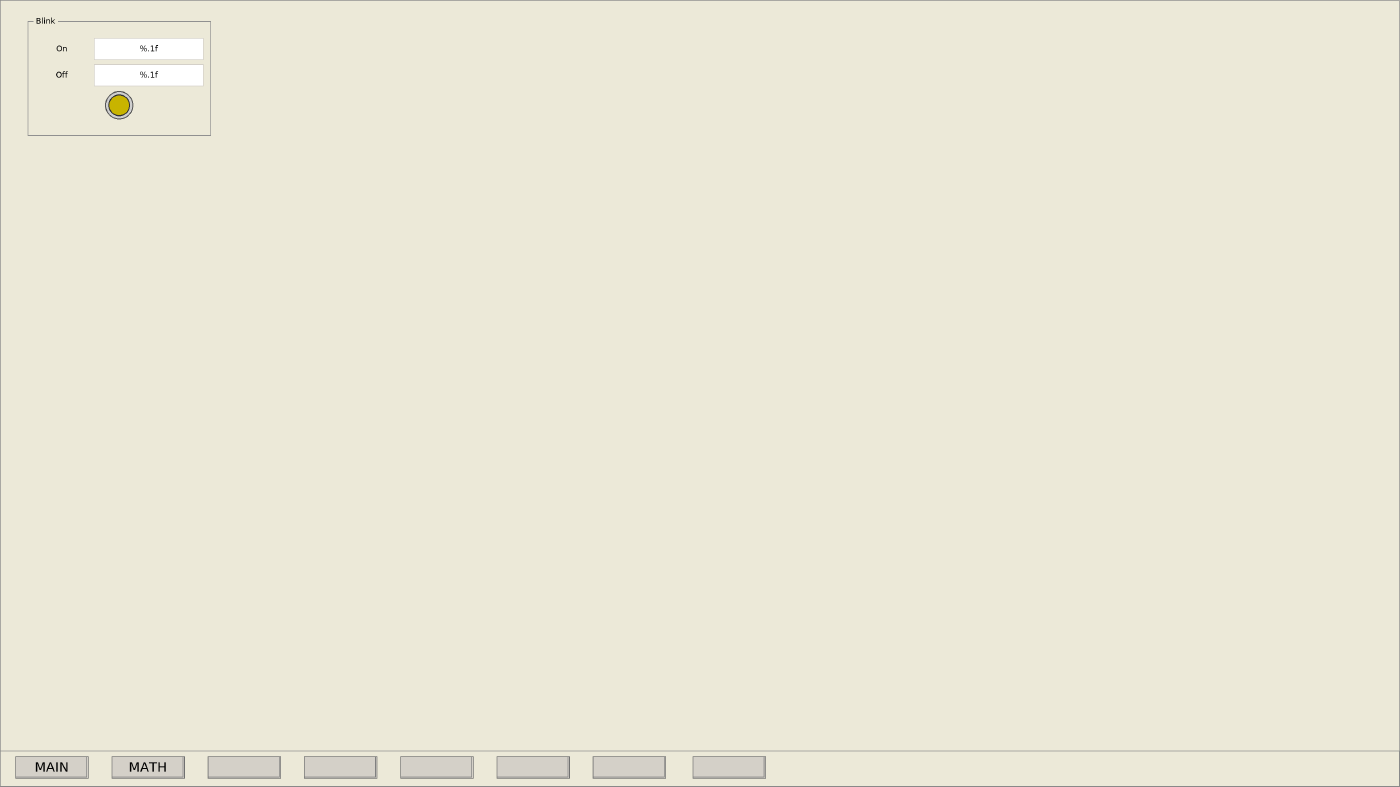
VISUALIZATION Visualization  // 1920x1080
    GroupBox (38,21 251x165), "Blink"
        Label (12,31 70x30), "On"
        Label (12,67 70x30), "Off"
        Lamp1 (103,101 45x45), variable: prgTestAuxsFuns.bOutputBlink, style: Lamp-Lamp1-Yellow
        Textfield (91,31 150x30), "%.1f", text variable: prgTestAuxsFuns.rBlinkOn
            OnMouseClick: write the text variable via Default
        Textfield (91,67 150x30), "%.1f", text variable: prgTestAuxsFuns.rBlinkOff
            OnMouseClick: write the text variable via Default
    Frame (0,1030 1920x50)
        shows Footer()
END_VISUALIZATION
